# EPICS autosave request: iocs/pylonIOC/iocBoot/iocPylon/auto_settings.req
file "pylon_settings.req",                P=$(P),  R=cam1:
file "NDStdArrays_settings.req",          P=$(P),  R=image1:
file "commonPlugin_settings.req",         P=$(P)
